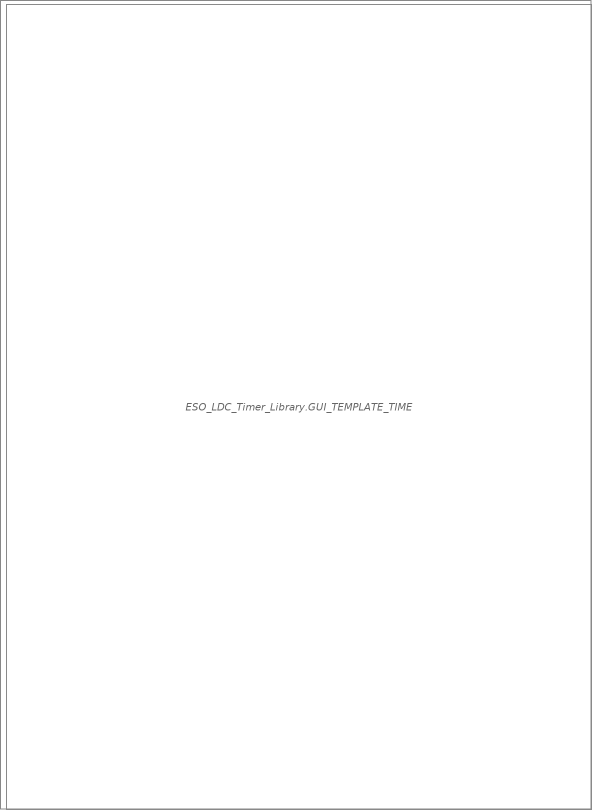
VISUALIZATION GUI_NOTT_TIME  // 592x810
    Frame (6,4 586x806)
        shows ESO_LDC_Timer_Library.GUI_TEMPLATE_TIME(m_DeviceName := 'NOTT Time', m_Instance := INFRATEC_TRIGERS.NottTime)
END_VISUALIZATION

(* stored: Version 1.1.0.1, ProductVersion 3.1.4024.12
   Visu GUI_NOTT_TIME: Id {30df6b72-9384-4599-871d-95cec70666e7} *)
